///////////
// Structure For I35. Main Operating Data to be saved (ex: OPC).  
//////////
TYPE PM_Standard :
STRUCT
		MesData						: PM ; (* Object *) 
	
END_STRUCT
END_TYPE

(* stored: Version 1.1.0.1, ProductVersion 3.1.4024.6
   DUT PM_Standard: Id {fa56d2c5-a27c-46fa-b5a8-6dc5213fe312} *)
